VAR_GLOBAL CONSTANT
    MAX_NUM_PIPER_MODULES : USINT := 100;
    MAI_NUM_PIPER_MODULES : USINT := MAX_NUM_PIPER_MODULES - 1;
END_VAR

(* stored: Version 1.1.0.1
   GVL PIPER_CONST: Id {07320410-48d8-43fe-bc90-eb7010206b8d} *)
